ABB RobotStudio station: Solution79.rspag

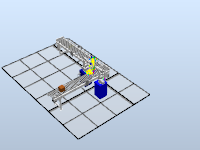
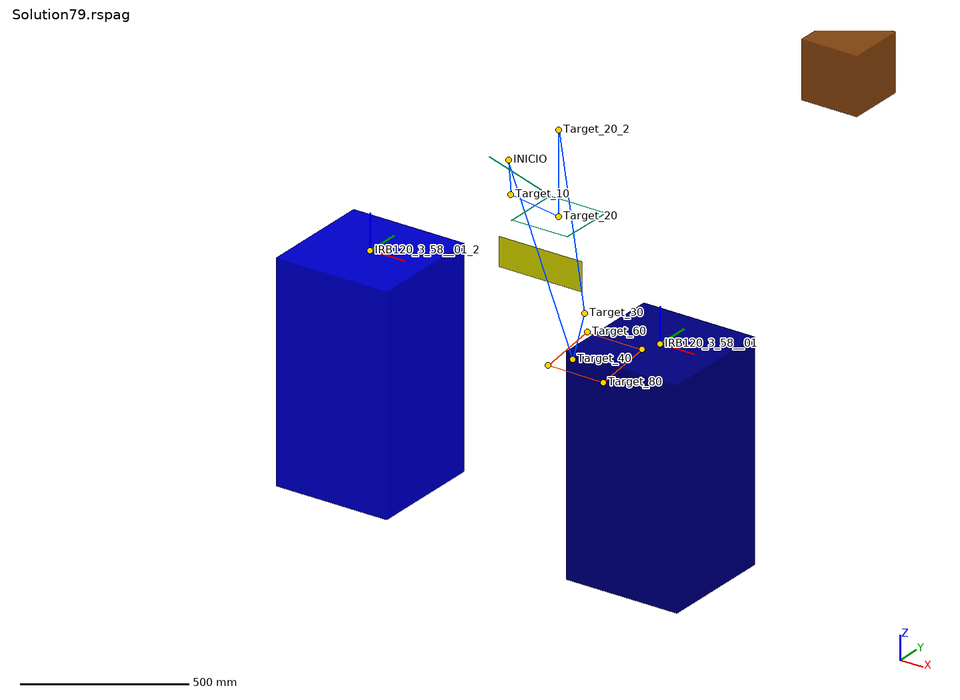
[picture v1: parts stored in the station drawn from their meshes, with robot base, taught points and paths (robot models come from the ABB library and are not in the file)]
--- station ---
Station Solution79 (saved by RobotStudio 21.2.9526.0)
Controller Controlador6, task T_ROB1: task frame (RAPID world) sits at (-614.53, 669.16, 750) mm in the station
Controller Controlador1, task T_ROB1: task frame (RAPID world) sits at (449.07, 645.97, 749.38) mm, rotated rx 0 ry 0 rz 180 deg in the station
Controller Controlador1
  mechanical unit ROB_1: IRB120_3_58__01, 6 joints, base frame (0, 0, 0) mm
Controller Controlador6
  mechanical unit ROB_1: IRB120_3_58__01_2, 6 joints, base frame (0, 0, 0) mm
Layout (positions relative to the parent item):
  - IRB120_3_58__01 [mechanism, from Robots\IRB120_3_58_G_01.rslib] at (449.07, 645.97, 749.38) mm, rotated rx 0 ry 0 rz 180 deg; joint values [0, 0, 0, 0, 0.5236, 0] (rad or m)
  - MyTool [mechanism, from Training Objects\myTool.rslib] at (84.72, 645.97, 1343.38) mm, rotated rx 180 ry 60 rz 0 deg
  - 400_guide [part, from Equipment\Conveyor Guide 400.rslib] at (177.98, -154.8, 0) mm, rotated rx 0 ry 0 rz 90 deg
  - 400_guide_2 [part, from Equipment\Conveyor Guide 400.rslib] at (3208.58, 252.55, 0) mm, rotated rx 0 ry 0 rz 180 deg
  - Soporte [part] at (249.07, 445.97, -0.62) mm, size 400 x 400 x 750 mm
  - Positioner_2 [smart component, from Components\Positioner.rslib] at (0, 0.42, 0) mm
      properties: Object=Caja; Position=[-0.113 2.176 0.784]; Orientation=[0 0 0]; Reference=Global; ReferenceObject=(none)
  - PlaneSensor [smart component, from Components\PlaneSensor.rslib] at (-162.05, 685.31, 817.94) mm, rotated rx 90 ry 0 rz 0 deg
      properties: Origin=[0 0 0]; Axis1=[0.3 0 0]; Axis2=[0 0.1 0]; SensedPart=(none)
    - _sensorPart_ [part], size 300 x 100 x 0 mm
  - PlaneSensor_2 [smart component, from Components\PlaneSensor.rslib] at (2142.88, 0.11, 996.88) mm, rotated rx 0 ry 90 rz 0 deg
      properties: Origin=[0 0 0]; Axis1=[0.1 0 0]; Axis2=[0 0.3 0]; SensedPart=(none)
    - _sensorPart_ [part], size 100 x 300 x 0 mm
  - SimulationEvents [smart component, from Components\SimulationEvents.rslib]
  - LogicSRLatch [smart component, from Components\LogicSRLatch.rslib]
  - LinearMover [smart component, from Components\LinearMover.rslib]
      properties: Object=Caja; Direction=[0 -0.1 0]; Speed=0.2; Reference=Global; ReferenceObject=(none)
  - Attacher [smart component, from Components\Attacher.rslib]
      properties: Parent=MyTool; Flange=0; Child=Caja; Mount=false; Offset=[0 0 0]; Orientation=[0 0 0]
  - Detacher [smart component, from Components\Detacher.rslib]
      properties: Child=Caja; KeepPosition=true
  - LogicSRLatch_2 [smart component, from Components\LogicSRLatch.rslib]
  - Componente inteligente_1 [smart component]
  - Caja [part] at (-113, 2176, 784) mm, size 200 x 200 x 200 mm
  - LinearMover_2 [smart component, from Components\LinearMover.rslib]
      properties: Object=Caja; Direction=[1 0 0]; Speed=0.2; Reference=Global; ReferenceObject=(none)
  - LogicGate_2 [smart component, from Components\LogicGate.rslib]
      properties: Operator=OR; Delay=1
  - Pieza_1 [part] at (-814.53, 469.16, 0) mm, size 400 x 400 x 750 mm
  - Pen [mechanism, from Training Objects\Pen.rslib] at (-250.18, 669.16, 1344) mm, rotated rx 180 ry 60 rz 180 deg
  - IRB120_3_58__01_2 [mechanism, from Robots\IRB120_3_58_G_01.rslib] at (-614.53, 669.16, 750) mm; joint values [0, 0, 0, 0, 0.5236, 0] (rad or m)
Attachment: MyTool is attached to IRB120_3_58__01 / Link6
Attachment: Pen is attached to IRB120_3_58__01_2 / Link6
Station signals: DI POSICIONADOR
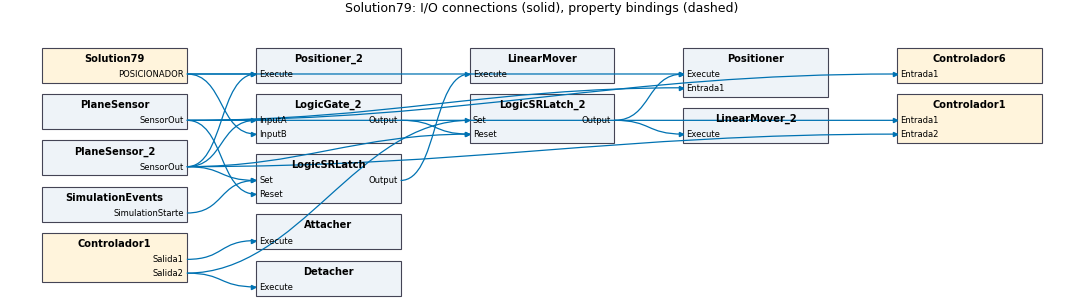
Station logic (signal -> signal, property => property):
  Solution79.POSICIONADOR -> Positioner.Execute
  Solution79.POSICIONADOR -> Positioner_2.Execute
  PlaneSensor.SensorOut -> Controlador1.Entrada1
  PlaneSensor_2.SensorOut -> Controlador1.Entrada2
  SimulationEvents.SimulationStarted -> LogicSRLatch.Set
  LogicSRLatch.Output -> LinearMover.Execute
  PlaneSensor.SensorOut -> LogicSRLatch.Reset
  Controlador1.Salida1 -> Attacher.Execute
  Controlador1.Salida2 -> Detacher.Execute
  LogicSRLatch_2.Output -> LinearMover_2.Execute
  Controlador1.Salida2 -> LogicSRLatch_2.Set
  LogicSRLatch_2.Output -> LinearMover_2.Execute
  PlaneSensor_2.SensorOut -> LogicGate_2.InputA
  LogicGate_2.Output -> LogicSRLatch_2.Reset
  Solution79.POSICIONADOR -> LogicGate_2.InputB
  PlaneSensor_2.SensorOut -> LogicSRLatch.Set
  PlaneSensor_2.SensorOut -> Positioner_2.Execute
  PlaneSensor_2.SensorOut -> LogicSRLatch_2.Reset
  PlaneSensor.SensorOut -> Controlador5.Entrada1
  PlaneSensor.SensorOut -> Controlador6.Entrada1
Targets, tools, work objects and paths stored in the station and not in the controller backup, written as RAPID:
! task T_ROB1
MODULE CalibData
  PERS tooldata Tooldata_1:=[TRUE,[[31.792631019,0,229.638935148],[0.945518576,0,0.325568154,0]],[1,[0,0,1],[1,0,0,0],0,0,0]];
  PERS tooldata Binzel:=[TRUE,[[123.560223674,0,296.652044776],[0.833885822,0,0.551936985,0]],[1,[0,0,100],[1,0,0,0],0,0,0]];
ENDMODULE

! task T_ROB1
MODULE Module1
  CONST robtarget posinic:=[[834.823430595,889.464897601,428.737205584],[0.183154359,-0.682483624,-0.683541371,-0.182870936],[-1,0,-1,0],[9E+09,9E+09,9E+09,9E+09,9E+09,9E+09]];
ENDMODULE


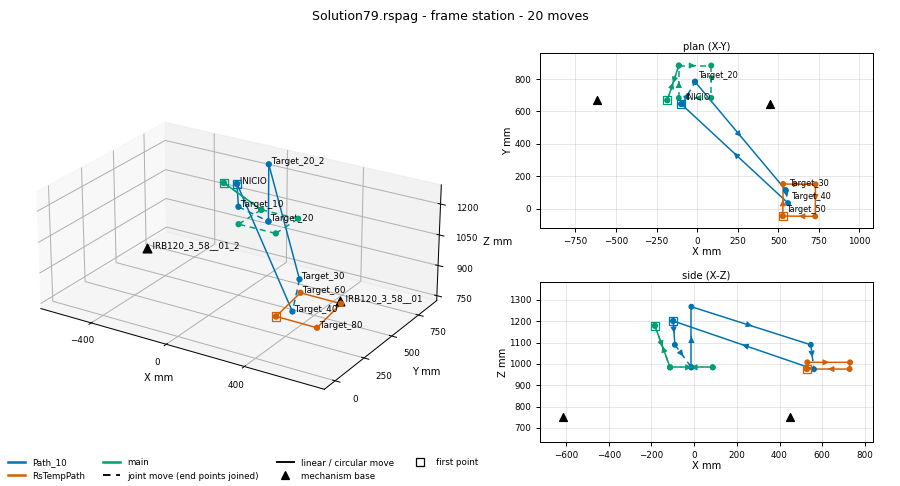
[picture p0: tool path of Solution79.rspag in frame station, 20 of 20 moves have a stored position in this frame; points joined in program order, loops and branches not executed]
--- Backups/Controlador1/RAPID/TASK1/PROGMOD/CalibData.mod ---
MODULE CalibData
    PERS tooldata MyTool:=[TRUE,[[31.792631019,0,229.638935148],[0.945518576,0,0.325568154,0]],[1,[0,0,1],[1,0,0,0],0,0,0]];
    TASK PERS wobjdata Workobject_Caja:=[FALSE,TRUE,"",[[0,0,0],[1,0,0,0]],[[0,0,0],[1,0,0,0]]];
ENDMODULE

--- Backups/Controlador1/RAPID/TASK1/PROGMOD/Module1.mod ---
MODULE Module1
        CONST robtarget INICIO:=[[547.330665099,0,451.647306311],[0.190808996,0,0.981627183,0],[0,-1,0,0],[9E+09,9E+09,9E+09,9E+09,9E+09,9E+09]];
    CONST robtarget Target_10:=[[539.367835409,0,340.165399999],[0.088323191,0,0.99609187,0],[-1,0,-1,0],[9E+09,9E+09,9E+09,9E+09,9E+09,9E+09]];
    CONST robtarget Target_20:=[[462.070173912,-137.232801189,234.618947582],[0.088323191,0,0.99609187,0],[0,0,0,0],[9E+09,9E+09,9E+09,9E+09,9E+09,9E+09]];
    CONST robtarget Target_30:=[[-97.269723866,530.524602292,340.165413516],[0.056542702,-0.765222972,0.637677676,0.067852108],[1,0,-1,0],[9E+09,9E+09,9E+09,9E+09,9E+09,9E+09]];
    CONST robtarget Target_40:=[[-112.033826088,611.733198811,225.637947582],[0,-0.707106781,0.707106781,0],[1,-1,0,0],[9E+09,9E+09,9E+09,9E+09,9E+09,9E+09]];
    CONST robtarget Target_50:=[[465.727415935,-0.168214349,479.273385052],[0.091553621,0.000179835,0.995800131,-0.000016534],[-1,-1,0,0],[9E+09,9E+09,9E+09,9E+09,9E+09,9E+09]];
    CONST robtarget Target_60:=[[371.063676927,281.449466007,479.273385052],[0.086776704,-0.317455729,0.943843098,0.029186802],[0,-1,-1,0],[9E+09,9E+09,9E+09,9E+09,9E+09,9E+09]];
    CONST robtarget Target_20_2:=[[462.070173912,-137.232801189,518.43482927],[0.088323191,0,0.99609187,0],[-1,0,-1,0],[9E+09,9E+09,9E+09,9E+09,9E+09,9E+09]];
!***********************************************************
    !
    ! Módulo:  Module1
    !
    ! Descripción:
    !   <Introduzca la descripción aquí>
    !
    ! Autor: raulb
    !
    ! Versión: 1.0
    !
    !***********************************************************


    !***********************************************************
    !
    ! Procedimiento Main
    !
    !   Este es el punto de entrada de su programa
    !
    !***********************************************************
    PROC main()
        !Añada aquí su código

        Path_10;
    ENDPROC
    PROC Path_10()
        INI:
        Setdo Salida1,0;
        Setdo Salida2,0;

        MoveL INICIO,v1000,fine,MyTool\WObj:=wobj0;
        WaitDI Entrada1,1;
         WaitTime 3;
        MoveL Target_10,v1000,fine,MyTool\WObj:=wobj0;
        MoveJdo Target_20,v200,z100,MyTool\WObj:=wobj0,Salida1,1;!atará la caja a la herramienta

        MoveL Target_20,v1000,z100,MyTool\WObj:=wobj0;
        MoveL Target_20_2,v500,fine,MyTool\WObj:=wobj0;
        MoveL Target_30,v1000,z100,MyTool\WObj:=wobj0;

        MoveJdo Target_40,v200,z100,MyTool\WObj:=wobj0,Salida2,1;!soltará la caja
        MoveL INICIO,v1000,fine,MyTool\WObj:=wobj0;
        WaitDI Entrada2,1;!espera al sensor 2
        WaitTime 2;
        GOTO INI;
    ENDPROC

ENDMODULE

--- Backups/Controlador1/RAPID/TASK1/PROGMOD/RsTempModule.mod ---
MODULE RsTempModule
    LOCAL CONST robtarget Target_50:=[[-79.157,690.849,226.711],[0,0.707106781,0.707106781,0],[0,0,0,0],[9E+09,9E+09,9E+09,9E+09,9E+09,9E+09]];
    LOCAL PERS tooldata MyTool:=[TRUE,[[31.7926,0,229.639],[0.945519,0,0.325568,0]],[1,[0,0,1],[1,0,0,0],0,0,0]];
    LOCAL PERS wobjdata Workobject_Caja:=[FALSE,TRUE,"",[[0,0,0],[1,0,0,0]],[[0,0,0],[1,0,0,0]]];
    LOCAL CONST robtarget Target_60:=[[-81.122,493.354,258.203],[0,0.707106781,0.707106781,0],[0,0,0,0],[9E+09,9E+09,9E+09,9E+09,9E+09,9E+09]];
    LOCAL CONST robtarget Target_70:=[[-281.112,495.301,257.935],[0,0.707106781,0.707106781,0],[0,0,0,0],[9E+09,9E+09,9E+09,9E+09,9E+09,9E+09]];
    LOCAL CONST robtarget Target_80:=[[-279.147,692.796,226.443],[0,0.707106781,0.707106781,0],[0,0,0,0],[9E+09,9E+09,9E+09,9E+09,9E+09,9E+09]];
PROC RsTempPath()
        MoveL Target_50,v1000,fine,MyTool\WObj:=Workobject_Caja;
        MoveL Target_60,v1000,fine,MyTool\WObj:=Workobject_Caja;
        MoveL Target_70,v1000,fine,MyTool\WObj:=Workobject_Caja;
        MoveL Target_80,v1000,fine,MyTool\WObj:=Workobject_Caja;
        MoveL Target_50,v1000,fine,MyTool\WObj:=Workobject_Caja;
ENDPROC

ENDMODULE

--- Backups/Controlador6/RAPID/TASK1/PROGMOD/CalibData.mod ---
MODULE CalibData
    PERS tooldata Pen_TCP:=[TRUE,[[110,0,140],[0.707106781,0,0.707106781,0]],[1,[10.7435139,0,140],[1,0,0,0],0,0,0]];
ENDMODULE

--- Backups/Controlador6/RAPID/TASK1/PROGMOD/Module1.mod ---
MODULE Module1
        CONST robtarget Target_10:=[[430.597385602,0,428.737205584],[0.258819045,0,-0.965925826,0],[0,0,0,0],[9E+09,9E+09,9E+09,9E+09,9E+09,9E+09]];
    CONST robtarget Target_20:=[[501.529,214.04,234],[0,0,1,0],[0,-2,1,0],[9E+09,9E+09,9E+09,9E+09,9E+09,9E+09]];
    CONST robtarget Target_30:=[[701.529,214.04,234],[0,0,1,0],[0,-2,1,0],[9E+09,9E+09,9E+09,9E+09,9E+09,9E+09]];
    CONST robtarget Target_40:=[[701.529,14.04,234],[0,0,1,0],[0,0,-1,1],[9E+09,9E+09,9E+09,9E+09,9E+09,9E+09]];
    CONST robtarget Target_50:=[[501.529,14.04,234],[0,0,1,0],[0,0,-1,1],[9E+09,9E+09,9E+09,9E+09,9E+09,9E+09]];
!***********************************************************
    !
    ! Módulo:  Module1
    !
    ! Descripción:
    !   <Introduzca la descripción aquí>
    !
    ! Autor: raulb
    !
    ! Versión: 1.0
    !
    !***********************************************************


    !***********************************************************
    !
    ! Procedimiento Main
    !
    !   Este es el punto de entrada de su programa
    !
    !***********************************************************
    PROC main()
        !Añada aquí su código
        INICIO:
        MoveL Target_10,v1000,z100,Pen_TCP\WObj:=wobj0;
        WaitDI Entrada1,1;
        MoveJ Target_20,v1000,fine,Pen_TCP\WObj:=wobj0;
        MoveJ Target_30,v1000,fine,Pen_TCP\WObj:=wobj0;
        MoveJ Target_40,v1000,fine,Pen_TCP\WObj:=wobj0;
        MoveJ Target_50,v1000,fine,Pen_TCP\WObj:=wobj0;
        MoveJ Target_20,v1000,fine,Pen_TCP\WObj:=wobj0;
        MoveL Target_10,v1000,fine,Pen_TCP\WObj:=wobj0;
        WaitTime 3;
        GOTO INICIO;

    ENDPROC
ENDMODULE

--- Backups/Controlador1/SYSPAR/EIO.cfg ---
EIO:CFG_1.0:6:1::
#
INDUSTRIAL_NETWORK:

      -Name "DeviceNet" -Label "DeviceNet Master/Slave Network" -Address "2"
#
DEVICENET_INTERNAL_DEVICE:

      -Name "DN_Internal_Device" -VendorName "ABB Robotics"\
      -ProductName "DeviceNet Internal Slave Device"
#
EIO_SIGNAL:

      -Name "Entrada1" -SignalType "DI" -Device "DN_Internal_Device"\
      -DeviceMap "0"

      -Name "Salida1" -SignalType "DO" -Device "DN_Internal_Device"\
      -DeviceMap "0"

      -Name "Entrada2" -SignalType "DI" -Device "DN_Internal_Device"\
      -DeviceMap "1"

      -Name "Salida2" -SignalType "DO" -Device "DN_Internal_Device"\
      -DeviceMap "1"

      -Name "Salida3" -SignalType "DO" -Device "DN_Internal_Device"\
      -DeviceMap "2"

--- Backups/Controlador6/SYSPAR/EIO.cfg ---
EIO:CFG_1.0:6:1::
#
INDUSTRIAL_NETWORK:

      -Name "DeviceNet" -Label "DeviceNet Master/Slave Network" -Address "2"
#
DEVICENET_INTERNAL_DEVICE:

      -Name "DN_Internal_Device" -VendorName "ABB Robotics"\
      -ProductName "DeviceNet Internal Slave Device"
#
EIO_SIGNAL:

      -Name "Entrada1" -SignalType "DI" -Device "DN_Internal_Device"\
      -DeviceMap "1"
